// TIA Portal V18 export
DATA_BLOCK "DB_CLOUD"   // DB1201
{ S7_Optimized_Access := 'FALSE' }
VERSION : 0.1
// stored: AutoNumber false, DBAccessibleFromOPCUA true, DBAccessibleFromWebserver true, IsOnlyStoredInLoadMemory false, IsWriteProtectedInAS false
   VAR
      P1S1O2 : Real := 1.0;
      P1S1CO2 : Real := 2.0;
      P1S1MT : Real := 3.0;
      P1S1H : Real := 4.0;
      P1S1PH : Real := 5.0;
      P1S2O2 : Real := 1.0;
      P1S2CO2 : Real := 2.0;
      P1S2MT : Real := 3.0;
      P1S2H : Real := 4.0;
      P1S2PH : Real := 5.0;
      P1S3O2 : Real := 1.0;
      P1S3CO2 : Real := 2.0;
      P1S3MT : Real := 3.0;
      P1S3H : Real := 4.0;
      P1S3PH : Real := 5.0;
      P2S1O2 : Real := 1.0;
      P2S1CO2 : Real := 2.0;
      P2S1MT : Real := 3.0;
      P2S1H : Real := 4.0;
      P2S1PH : Real := 5.0;
      P2S2O2 : Real := 1.0;
      P2S2CO2 : Real := 2.0;
      P2S2MT : Real := 3.0;
      P2S2H : Real := 4.0;
      P2S2PH : Real := 5.0;
      P2S3O2 : Real := 1.0;
      P2S3CO2 : Real := 2.0;
      P2S3MT : Real := 3.0;
      P2S3H : Real := 4.0;
      P2S3PH : Real := 5.0;
      P3S1O2 : Real := 1.0;
      P3S1CO2 : Real := 2.0;
      P3S1MT : Real := 3.0;
      P3S1H : Real := 4.0;
      P3S1PH : Real := 5.0;
      P3S2O2 : Real := 1.0;
      P3S2CO2 : Real := 2.0;
      P3S2MT : Real := 3.0;
      P3S2H : Real := 4.0;
      P3S2PH : Real := 5.0;
      P3S3O2 : Real := 1.0;
      P3S3CO2 : Real := 2.0;
      P3S3MT : Real := 3.0;
      P3S3H : Real := 4.0;
      P3S3PH : Real := 5.0;
      P4S1O2 : Real := 1.0;
      P4S1CO2 : Real := 2.0;
      P4S1MT : Real := 3.0;
      P4S1H : Real := 4.0;
      P4S1PH : Real := 5.0;
      P4S2O2 : Real := 1.0;
      P4S2CO2 : Real := 2.0;
      P4S2MT : Real := 3.0;
      P4S2H : Real := 4.0;
      P4S2PH : Real := 5.0;
      P4S3O2 : Real := 1.0;
      P4S3CO2 : Real := 2.0;
      P4S3MT : Real := 3.0;
      P4S3H : Real := 4.0;
      P4S3PH : Real := 5.0;
      P5S1O2 : Real := 1.0;
      P5S1CO2 : Real := 2.0;
      P5S1MT : Real := 3.0;
      P5S1H : Real := 4.0;
      P5S1PH : Real := 5.0;
      P5S2O2 : Real := 1.0;
      P5S2CO2 : Real := 2.0;
      P5S2MT : Real := 3.0;
      P5S2H : Real := 4.0;
      P5S2PH : Real := 5.0;
      P5S3O2 : Real := 1.0;
      P5S3CO2 : Real := 2.0;
      P5S3MT : Real := 3.0;
      P5S3H : Real := 4.0;
      P5S3PH : Real := 5.0;
      P6S1O2 : Real := 1.0;
      P6S1CO2 : Real := 2.0;
      P6S1MT : Real := 3.0;
      P6S1H : Real := 4.0;
      P6S1PH : Real := 5.0;
      P6S2O2 : Real := 1.0;
      P6S2CO2 : Real := 2.0;
      P6S2MT : Real := 3.0;
      P6S2H : Real := 4.0;
      P6S2PH : Real := 5.0;
      P6S3O2 : Real := 1.0;
      P6S3CO2 : Real := 2.0;
      P6S3MT : Real := 3.0;
      P6S3H : Real := 4.0;
      P6S3PH : Real := 5.0;
   END_VAR
BEGIN
END_DATA_BLOCK
